// Mitsubishi GX Works2 project: FUNCTION BLOCK   PLC: Q03UDV

// task Task_01 (event TRUE, interval 0, priority 31): POU_01

PROGRAM POU_01
VAR
  CTD_1 : CTD;
  CTD1 : BOOL;
  CTU_1 : CTU;
  R_TRIG_1 : R_TRIG;
  CTUD_1 : CTUD;
  CTUD_2 : CTUD;
  TP_1 : TP;
  TON_1 : TON;
  TOF_1 : TOF;
  TimeTP : TIME;
  TimeTN : TIME;
  TimeTF : TIME;
  TP_2 : TP;
END_VAR
(* structured ladder/FBD written out as ST: instructions are called as NAME(EN, inputs, outputs); _pN, _eN, _tN stand for wires *)
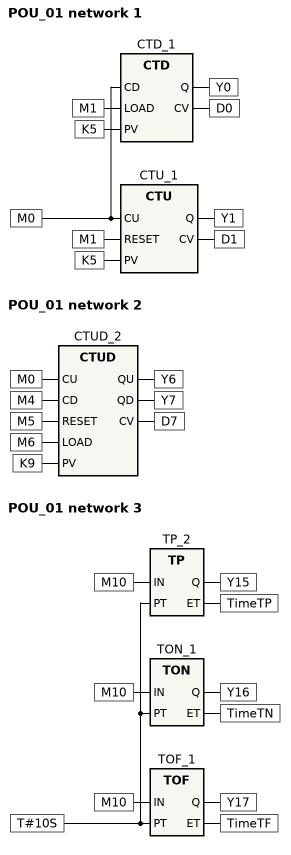
(* network 1 *)
CTD_1(CD := M0, LOAD := M1, PV := K5, Q => Y0, CV => D0);
CTU_1(CU := M0, RESET := M1, PV := K5, Q => Y1, CV => D1);
(* network 2 *)
CTUD_2(CU := M0, CD := M4, RESET := M5, LOAD := M6, PV := K9, QU => Y6, QD => Y7, CV => D7);
(* network 3 *)
TP_2(IN := M10, PT := T#10S, Q => Y15, ET => TimeTP);
TON_1(IN := M10, PT := T#10S, Q => Y16, ET => TimeTN);
TOF_1(IN := M10, PT := T#10S, Q => Y17, ET => TimeTF);
END_PROGRAM
